(* IEC 61131-3 sources: repolevel_ST_code_completion/output/0127完整版本_带planner/repoeval_GreatExampleOfAdvantages/readful_result, 2 files *)

(* ---- Home.st ---- *)
FUNCTION_BLOCK Home
VAR_INPUT
END_VAR
VAR_OUTPUT
END_VAR
VAR
    InternalState: INT;
    GroundFloorState: INT;
    TopFloorState: INT;
    MQTTMessage: STRING;
END_VAR

// GroundFloor and TopFloor function calls removed because they are not defined.
// GroundFloor();
// TopFloor();

IF InternalState = 0 THEN
// Replace undefined GroundFloor and TopFloor references with placeholder static values.
  GroundFloorState := 0; // Placeholder value since GroundFloor.LivingRoom.LampXOut is not defined.
  TopFloorState := 0;    // Placeholder value since TopFloor.MainBath.LampXOut is not defined.
    InternalState := 1;
END_IF

IF InternalState = 1 THEN
    IF GroundFloorState > 0 THEN
        MQTTMessage := 'Ground Floor Active';
    ELSIF TopFloorState > 0 THEN
        MQTTMessage := 'Top Floor Active';
    ELSE
        MQTTMessage := 'No Activity';
    END_IF
    InternalState := 2;
END_IF

IF InternalState = 2 THEN
    // Simulate sending MQTT message
// MQTT.CallbackCollector is not defined. Replace with a placeholder or comment.
  // Simulate sending MQTT message process here.
    InternalState := 3;
END_IF

IF InternalState = 3 THEN
    // Reset states for next operation
    GroundFloorState := 0;
    TopFloorState := 0;
    InternalState := 0;
END_IF
END_FUNCTION_BLOCK

(* ---- MQTT_STUFF.st ---- *)
FUNCTION_BLOCK MQTT_STUFF
VAR_INPUT
END_VAR
VAR_OUTPUT
END_VAR
VAR
    connectionStatus: BOOL;
    reconnectTimer: TON;
    messageReceived: BOOL;
    receivedMessage: STRING(255);
END_VAR

IF NOT init THEN
    init := TRUE;
    Subscriber.SetMqttInOut(MQTT_IN_OUT := GVL_MQTT.MQTT_IN_OUT);
    SubscribeTopic := InstanceName.GetInstanceTopic();
    birthTopic := SubscribeTopic;
    found := CommonTypesAndFunctions.find(str1 := ADR(SubscribeTopic), str2 := ADR('/'));
    found := found + 1 + CommonTypesAndFunctions.find(str1 := ADR(SubscribeTopic[found + 1]), str2 := ADR('/'));
    pt := ADR(SubscribeTopic[found + 1]);
    pt^ := 'Receive/#';
    GVL_MQTT.MQTT_IN_OUT.ClientID := CONCAT('CodesysMqtt', TO_STRING(TICKS.GetTick(xDummy := TRUE)));
END_IF

GVL_MQTT.MQTT_IN_OUT.clientFB(
    MQTT_IN_OUT := GVL_MQTT.MQTT_IN_OUT,
    xConnect := TRUE,
    xDisconnect := FALSE,
    xPublish := FALSE,
    xSubscribe := TRUE,
    xUnsubscribe := FALSE
);

connectionStatus := GVL_MQTT.MQTT_IN_OUT.clientFB.xConnected;

connectRising(CLK := connectionStatus);

IF connectRising.Q THEN
    birthMessage.SetMqttInOut(MQTT_IN_OUT := GVL_MQTT.MQTT_IN_OUT);
    birthMessage.SetTopic(Topic := birthTopic);
    birthMessage.SetPayload(Payload := 'Device Online');
    birthMessage.Publish();
END_IF

Subscriber.Subscribe(Topic := SubscribeTopic);

messageReceived := Subscriber.GetMessage(Topic := SubscribeTopic, Payload := receivedMessage);

IF messageReceived THEN
    // Handle received message (e.g., pass to Collector callback mechanism)
    xxx := ADR(receivedMessage);
END_IF

reconnectTimer(IN := NOT connectionStatus, PT := T#10S);

IF reconnectTimer.Q THEN
    GVL_MQTT.MQTT_IN_OUT.clientFB.xConnect := TRUE;
END_IF
END_FUNCTION_BLOCK
